FUNCTION_BLOCK AlbertsContext EXTENDS TcoCore.TcoContext
VAR
	Machine : AlbertsMachine(THIS^);
END_VAR

(*~
	<docu>
		<summary>
			Main method of the TcoContext. This is the entry point of any control logic that belongs to this context. 
			The call of this method is ensured by calling the <c>InstanceName.Run()</c> method, and it must not be called explicitly.
			This method is abstract, and it must be overridden in derived block.
		</summary>
	</docu>
~*)
METHOD PROTECTED  Main
Machine();
END_METHOD

END_FUNCTION_BLOCK

(* stored: Version 1.1.0.1, ProductVersion 3.1.4024.5
   POU AlbertsContext: Id {77d39940-ac26-0912-24b5-a04540c6369c}, SpecialFunc None
   Method Main: Id {b613b3f3-a147-0c50-1f7d-e0378b0d00f9} *)
